Fanuc TP program (LS listing): ZERO_R01.LS

/PROG  ZERO_R01
/ATTR
OWNER		= MNEDITOR;
COMMENT		= "Alias -> GO_ZERO_R01";
PROG_SIZE	= 0;
CREATE		= DATE 08-10-07  TIME 00:28:06;
MODIFIED	= DATE 26-04-20  TIME 12:00:00;
FILE_NAME	= ;
VERSION		= 0;
LINE_COUNT	= 3;
MEMORY_SIZE	= 0;
PROTECT		= READ_WRITE;
STORAGE		= SHADOW;
TCD:  STACK_SIZE	= 0,
      TASK_PRIORITY	= 50,
      TIME_SLICE	= 0,
      BUSY_LAMP_OFF	= 0,
      ABORT_REQUEST	= 0,
      PAUSE_REQUEST	= 0;
DEFAULT_GROUP	= 1,*,*,*,*;
CONTROL_CODE	= 00000000 00000000;
/APPL

AUTO_SINGULARITY_HEADER;
  ENABLE_SINGULARITY_AVOIDANCE   : TRUE;

LINE_TRACK;
  LINE_TRACK_SCHEDULE_NUMBER      : 0;
  LINE_TRACK_BOUNDARY_NUMBER      : 0;
  CONTINUE_TRACK_AT_PROG_END      : TRUE;

/MN
   1:  !ALIAS -- DELEGATES TO GO_ZERO_R01 ;
   2:  !(kept so legacy callers don't break) ;
   3:  CALL GO_ZERO_R01    ;
/POS
/END
